// TIA Portal V20 export
// export: Created 2026-10-03T18:54:34.7942104Z, ExportSetting WithDefaults, DisplayName Totally Integrated Automation Portal, DisplayVersion V20 Update 4, DisplayName TIA Portal Openness, DisplayVersion V20 Update 4, DisplayName TIA Portal Version Control Interface, DisplayVersion V20 Update 4, DisplayName SINAMICS Startdrive Advanced, DisplayVersion V20 SP1 Update 1, DisplayName SINAMICS Startdrive G110M, G120, G120C, G120D, G120P, G115D, DisplayVersion V20 SP1 Update 1, DisplayName SINAMICS Startdrive G130, G150, S120, S150, SINAMICS MV, G220, S200, S210, DisplayVersion V20 SP1 Update 1, DisplayName STEP 7 Professional, DisplayVersion V20 Update 4, DisplayName STEP 7 Safety, DisplayVersion V20 Update 2, DisplayName WinCC Basic/Comfort/Advanced, DisplayVersion V20 Update 4, DisplayName WinCC Unified, DisplayVersion V20 Update 4
FUNCTION "SLC_TO_TIME" : Time   // FC23, SCL
TITLE = SLC timer counts to TIME
{ S7_Optimized_Access := 'TRUE' }
VERSION : 0.1
// Converts an SLC timer value (counts of the timer's timebase) to a TIA TIME.
//  Used where SLC logic moved a calculated word into a timer preset (MOV N7:x T4:y.PRE).
// stored: AutoNumber true, IsIECCheckEnabled false, SetENOAutomatically false, UDAEnableTagReadback false
   VAR_INPUT
      Counts : Int;   // Value in timebase counts, as the SLC stored it
      BaseMs : DInt;   // Timebase in milliseconds: 1000 for 1.0 s, 10 for 0.01 s, 1 for 0.001 s
   END_VAR
BEGIN
   // TIME counts milliseconds, so the counts only need scaling by the timebase.
   #SLC_TO_TIME := DINT_TO_TIME(INT_TO_DINT(#Counts) * #BaseMs);
END_FUNCTION
